DATA_BLOCK "DB1"
{ S7_Optimized_Access := 'FALSE' }
VERSION : 0.1
NON_RETAIN
   STRUCT
      DF : Bool;
      FF : Bool;
      GH : Bool;
      JJ : Bool;
      LL : Int;
      II : Int;
   END_STRUCT;


BEGIN

END_DATA_BLOCK

